Universal Robots PolyScope program: rtde_depowdering.urp

Program rtde_depowdering (installation=default directory=/programs/usbdisk/depowdering createdIn=3.2.19275.0 lastSavedIn=5.12.0.1101482 robotSerialNumber=20225501047)
Calibrated DH parameters: a=[0.000165, -0.414236, -0.366713, 0.000028, 0.000067, 0]; d=[0.162801, -57.2398, 32.079015, 25.294245, 0.099708, 0.099569]; alpha=[1.570474, 0.001669, 0.005558, 1.570315, -1.568415, 0]; deltaTheta=[0, -0.226697, 6.145588, 0.364296, 0.000001, 0]
BeforeStart
  setp := get_actual_joint_positions()
  Script: write_output_integer_register(0,1)
  Wait Sleep waitTime=0.01
  Popup Message (haltProgram=false message=Initialized inputType=Text)
Robot Program (runOnlyOnce=false)
  Script: write_output_integer_register(0, 1)
  Script: sync()
  MoveL speed 250 mm/s, acceleration 1200 mm/s^2 (useActiveTCP=true) feature=Base
    Waypoint Waypoint (Variable): variable=setp
  Script: write_output_integer_register(0, 0)
  Loop While (checkContinuously=false) expression=read_input_integer_register(0)≟1
    Script: sync()
  Script: write_output_integer_register(0,1)
  Script: sync()
Thread Thread_1 (runOnlyOnce=false)
  Loop Forever
    tmp := p[0,0,0,0,0,0]
    Script: tmp[0] = read_input_float_register(0)
    Script: tmp[1] = read_input_float_register(1)
    Script: tmp[2] = read_input_float_register(2)
    Script: tmp[3] = read_input_float_register(3)
    Script: tmp[4] = read_input_float_register(4)
    Script: tmp[5] = read_input_float_register(5)
    setp := get_inverse_kin(p[tmp[0],tmp[1],tmp[2],tmp[3],tmp[4],tmp[5]],get_actual_joint_positions())
    Script: sync()
